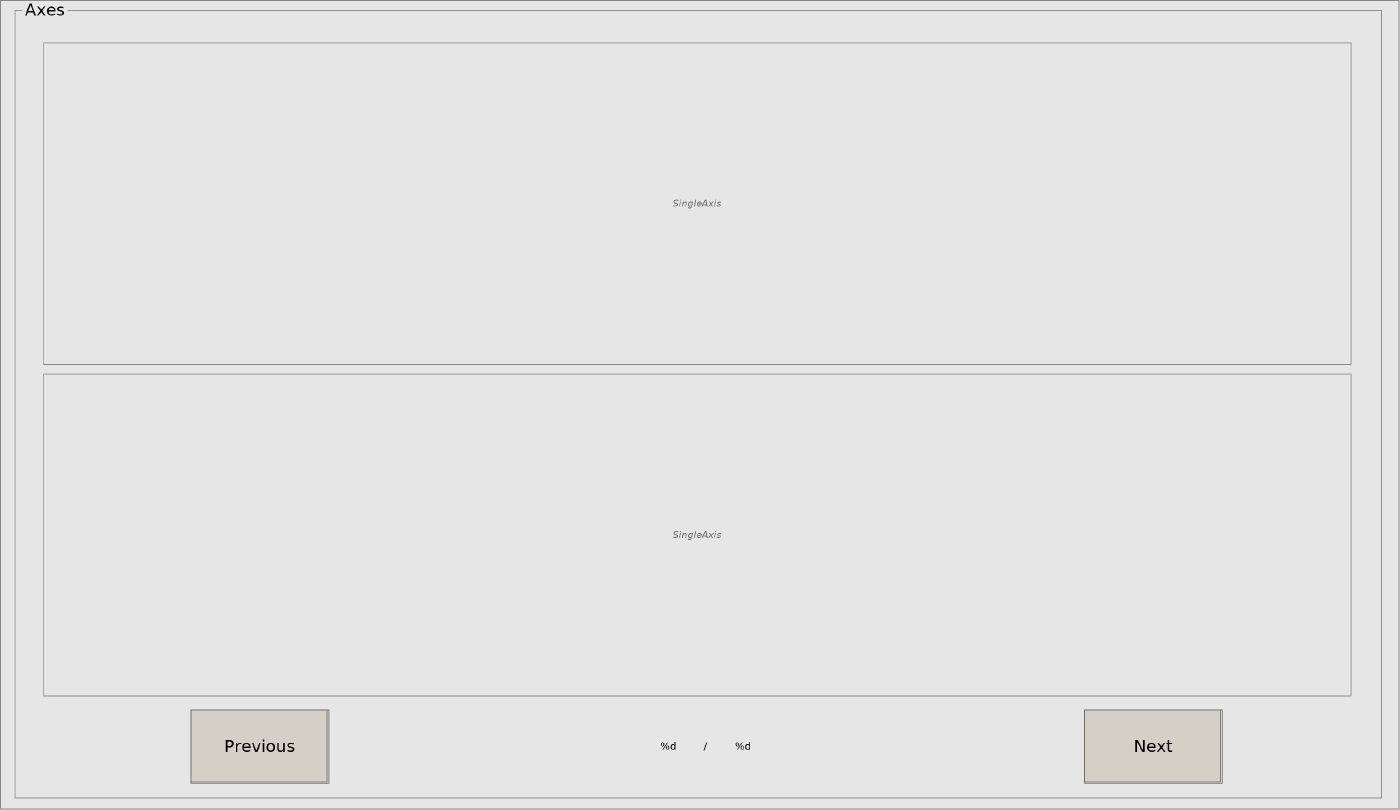
VISUALIZATION PageManualAxis_1  // 1520x880
VAR_IN_OUT
	btnPrevious			: BOOL;
	btnNext				: BOOL;
	bPreviousInvisible	: BOOL;
	bNextInvisible		: BOOL;
	stAxisEmpty			: ARRAY[0..1] OF BOOL;
	stAxis				: ARRAY[0..1] OF ST_VisuCtrlAxisFrame;
	iAxisSelectedPageIndex		: USINT;
	iAxisTotalPageIndex 		: USINT;
END_VAR
    GroupBox (16,3 1484x864), "Axes"
        Frame (31,43 1420x350), invisible if: stAxisEmpty[0]
            shows SingleAxis(stAxis := stAxis[0])
        Button (1161,768 150x80), "Next", invisible if: bNextInvisible
            tap btnNext
        Button (191,768 150x80), "Previous", invisible if: bPreviousInvisible
            tap btnPrevious
        Frame (31,403 1420x350), invisible if: stAxisEmpty[1]
            shows SingleAxis(stAxis := stAxis[1])
        Rectangle (685,783 130x50), "/"
        Rectangle (685,783 50x50), "%d", text variable: iAxisSelectedPageIndex+1
        Rectangle (766,783 50x50), "%d", text variable: iAxisTotalPageIndex+1
END_VISUALIZATION

(* stored: Version 1.1.0.1, ProductVersion 3.1.4024.12
   Visu PageManualAxis_1: Id {b3a37902-1a88-4bcd-af20-eeafbd1b0d56} *)
